PROGRAM MODE_SELECTION_1
VAR
	//MagnetState : (FULL_SHUTDOWN, IDLE, READY_TO_CHARGE, CHARGING, CHARGING_PAUSED, READY_TO_SHOOT, SHOOTING, POST_SHOT, SHUTDOWN, DUMPING); 
	eMagState : E_MagState := 0;
	//bChargingDone: BOOL;
	eCommand : E_Command; // Requested State (FULL_SHUT_DOWN = 0, IDLE = 1, CHARGE = 2, CHARGE_PAUSED, SHOOT = 3, POST_SHOT = 4, SHUTDOWN = 5, DUMPING = 6)
	eStatus : E_Status; // Actual Status (FULL_SHUTDOWN = 0, IDLE = 1, READY_TO_CHARGE = 2, CHARGE = 3, CHARGE_PAUSED = 4, READY_TO_SHOOT = 5, SHOOTING = 6, POST_SHOT = 7, SHUTDOWN = 8, DUMPING = 9, TRIPPED = 10, MANUAL_MODE = 11)
	i: INT;
	
	ChargerOFF_ChrgRlyOPEN_Delay_FShutDown_TON	: TON;
	timerBTW_ChrgRly_ChrgEnable_ChrgPause_TON	: TON;
	timerBTW_ChrgRly_ChrgEnable_ReadyToShoot_TON: TON;
	
	timerBTW_ChrgRly_ChrgEnable_Chrging_TON		: TON;
	timerBTW_ChrgRly_ChrgEnable_PT 	: TIME := T#500MS;
	timerBTW_ChrgRly_ChrgEnable_ET  : TIME;
	
	timerBTW_DUMP_IDLE 				: TON;
	timerBTW_DUMP_IDLE_PT 			: TIME := T#15S;
	timerBTW_DUMP_IDLE_ET 			: TIME;
	
	timerForChargertoTurnOn_TON		: TON;
	timerForChargertoTurnOn_PT		: TIME := T#10S;
	timerForChargertoTurnOn_ET		: TIME;
	ChargersReady					: BOOL;
	
	timerBTW_Shoot_PostShot_TON		: TON;
	timerBTW_Shoot_PostShot_PT      : TIME := T#2S;
	timerBTW_Shoot_PostShot_ET		: TIME;
	
	timerBTW_ChrgEnable_ChrgRly_ShutDown_TON	: TON;
	timerBTW_ChrgEnable_ChrgRly_PT				: TIME := T#1S;
	timerBTW_ChrgEnable_ChrgRly_ET				: TIME;
	
	timerBTW_ChrgEnable_ChrgRly_Dumping_TON		: TON;
	timerBTW_ChrgEnable_ChrgRly_Dumping_ET		: TIME;
	
	timerBTW_ChrgEnable_ChrgRly_Tripped_TON		: TON;
	timerBTW_ChrgEnable_ChrgRly_Tripped_ET		: TIME;
	
	ReadyToChargeRunOutTMR_TON					: TON;
	ReadyToChargeRunOutTMR_PT					: TIME := T#1200S;
	ReadyToChargeRunOutTMR_ET					: TIME;
	
	ChargePausedRunOutTMR_TON					: TON;
	ChargePausedRunOutTMR_PT					: TIME := T#30S;
	ChargePausedRunOutTMR_ET					: TIME;
	
	ReadyToShootRunOutTMR_TON					: TON;
	ReadyToShootRunOutTMR_PT					: TIME := T#60S;
	ReadyToShootRunOutTMR_ET					: TIME;
	
	ShootingRunOutTMR_TON						: TON;
	ShootingRunOutTMR_PT						: TIME := T#3S;
	ShootingRunOutTMR_ET						: TIME;
	
	PostShotRunOutTMR_TON						: TON;
	PostShotRunOutTMR_PT						: TIME := T#2S;
	PostShotRunOutTMR_ET						: TIME;
	
	DumpingRunOutTMR_TON						: TON;
	DumpingRunOutTMR_PT							: TIME := T#300S;
	DumpingRunOutTMR_ET							: TIME;
	
	ChargingRunOutTMR_TON						: TON;
	ChargingRunOutTMR_PT						: TIME := T#600S;
	ChargingRunOutTMR_ET						: TIME;
	
	stControl									: ST_Control;
END_VAR


//LCP Indicator for charged/charging
FOR i := 1 TO 10 BY 1 DO
	IF ( Devices.Coil[i].ChargeRelay_closed = TRUE AND 
		Devices.Coil[i].CoilEnabled = TRUE AND 
		Devices.Coil[i].enableOutputToCharger = TRUE ) OR Devices.Coil[i].ChargeVoltageFeedback >= 10
	THEN
		Devices.Coil[i].SystemCharging := TRUE;
		ELSE
			Devices.Coil[i].SystemCharging := FALSE;
	END_IF;
END_FOR;

//IF any one of the systems is charging or charge, then all system discharge is false, otherwise true
IF Devices.Coil[i].SystemCharging = TRUE THEN
	GVL.AllSystemsDischarged := FALSE;
ELSE
	GVL.AllSystemsDischarged := TRUE;
END_IF;

// IF system is tripped at anytime, it goes to tripped state
IF Trips_DB.SystemTripped = TRUE OR Permissives_DB.SafetyOK = FALSE THEN
	eMagState := E_MagState.TRIPPED;
END_IF;

IF MCP_IO.RemoteModeSelected = FALSE OR HMI_DB.RemoteModeSelected = FALSE THEN  //change auto to remote / manu to local
	eStatus := E_Status.MANUAL_MODE;
END_IF

//At any point, if screen room ask to dump, it goes to dump state
IF (MCP_IO.RemoteModeSelected = TRUE AND eCommand = E_Command.DUMP) OR stControl.Abort = TRUE THEN
	eMagState := E_Magstate.DUMPING;
END_IF;

FOR i := 1 TO 10 BY 1 DO
	Devices.Coil[i].NumOfCap := Tx_Config.CoilSP[i].SysParameters.NumOfCaps;
END_FOR


//Process Starts
CASE eMagState OF 
	//Full Shutdown
	E_MagState.FULL_SHUTDOWN:
						//Disable all Chargers
						FOR i := 1 TO 10 BY 1 DO
							
							//open (de-energize) all interlock relays
							Devices.Coil[i].CloseACInterlockRly := FALSE;
							Devices.Coil[i].enableOutputToCharger := FALSE;
			
							//Close (de-energize) All Dump relays
							Devices.Coil[i].OpenDumpRelays := FALSE;
							
							Devices.Coil[i].CloseHVisolationRelay := FALSE;   //Open all HV isolation relays
						END_FOR;
						
						ChargerOFF_ChrgRlyOPEN_Delay_FShutDown_TON (IN:=TRUE, PT:= timerBTW_ChrgRly_ChrgEnable_PT);
						//delay 500ms before opening charge relay
						IF ChargerOFF_ChrgRlyOPEN_Delay_FShutDown_TON.Q = TRUE THEN
							FOR i := 1 TO 10 BY 1 DO		
							//open (de-energize) all interlock relays
							Devices.Coil[i].closeChargeRelay := FALSE;	
							END_FOR;
							ChargerOFF_ChrgRlyOPEN_Delay_FShutDown_TON (IN:=FALSE, PT:= timerBTW_ChrgRly_ChrgEnable_PT);
						END_IF;
						
						//send shutdown status to screen room
						eStatus := E_Status.FULL_SHUTDOWN;
						//if auto mode selected or hmi automode is selected and screen room asks for idle mode go to idle mode
						IF (MCP_IO.RemoteModeSelected = TRUE OR HMI_DB.RemoteModeSelected = TRUE) AND eCommand = E_Command.IDLE THEN //Auto mode
							GVL.fullshutdown_to_idle := TRUE;
							//if in manu mode and safety is okay and HMI idle MODE PB is pressed, go to idle mode
						ELSIF HMI_DB.RemoteModeSelected = FALSE AND Permissives_DB.SafetyOK = TRUE AND HMI_DB.Idle_mode = TRUE THEN //Manu mode
							GVL.fullshutdown_to_idle := TRUE;
						ELSE
							GVL.fullshutdown_to_idle := FALSE; // otherwise do nothing.
						END_IF;
	
						IF GVL.fullshutdown_to_idle = TRUE THEN
							eMagState := E_MagState.IDLE;
						END_IF;
						//reset all run out tmr
						ReadyToChargeRunOutTMR_TON (IN := FALSE, PT := ReadyToChargeRunOutTMR_PT, ET=>ReadyToChargeRunOutTMR_ET);
						ChargingRunOutTMR_TON (IN := FALSE, PT := ChargingRunOutTMR_PT, ET => ChargingRunOutTMR_ET);
						ChargePausedRunOutTMR_TON (IN := FALSE, PT := ChargePausedRunOutTMR_PT, ET=> ChargePausedRunOutTMR_ET);
						ReadyToShootRunOutTMR_TON (IN := FALSE, PT := ReadyToShootRunOutTMR_PT, ET => ReadyToShootRunOutTMR_ET);
						ShootingRunOutTMR_TON (IN := FALSE, PT := ShootingRunOutTMR_PT, ET => ShootingRunOutTMR_ET);
						PostShotRunOutTMR_TON (IN := FALSE, PT := PostShotRunOutTMR_PT, ET => PostShotRunOutTMR_ET);
						DumpingRunOutTMR_TON (IN := FALSE, PT := DumpingRunOutTMR_PT, ET => DumpingRunOutTMR_ET);
		
	//IDLE STATE
	E_MagState.IDLE:
						eStatus := E_Status.IDLE; //Send status state to screen room
						GVL.dump_to_idle := FALSE;
						//reset all run out tmr
						ReadyToChargeRunOutTMR_TON (IN := FALSE, PT := ReadyToChargeRunOutTMR_PT, ET=>ReadyToChargeRunOutTMR_ET);
						ChargingRunOutTMR_TON (IN := FALSE, PT := ChargingRunOutTMR_PT, ET => ChargingRunOutTMR_ET);
						ChargePausedRunOutTMR_TON (IN := FALSE, PT := ChargePausedRunOutTMR_PT, ET=> ChargePausedRunOutTMR_ET);
						ReadyToShootRunOutTMR_TON (IN := FALSE, PT := ReadyToShootRunOutTMR_PT, ET => ReadyToShootRunOutTMR_ET);
						ShootingRunOutTMR_TON (IN := FALSE, PT := ShootingRunOutTMR_PT, ET => ShootingRunOutTMR_ET);
						PostShotRunOutTMR_TON (IN := FALSE, PT := PostShotRunOutTMR_PT, ET => PostShotRunOutTMR_ET);
						DumpingRunOutTMR_TON (IN := FALSE, PT := DumpingRunOutTMR_PT, ET => DumpingRunOutTMR_ET);
						
						// Local MODE
						IF (MCP_IO.RemoteModeSelected = FALSE OR HMI_DB.RemoteModeSelected = FALSE)AND 
							HMI_DB.chargePB = TRUE AND 
							Permissives_DB.SafetyOK = TRUE AND 
							GVL.AllSystemsDischarged = TRUE 
							THEN   
								//open dump relays
								FOR i := 1 TO 10 BY 1 DO
									Devices.Coil[i].OpenDumpRelays := TRUE; //NC contact
								END_FOR;
			
								GVL.idle_to_readyToCharge := TRUE;
							ELSE
								GVL.idle_to_readyToCharge := FALSE;
						END_IF;
						//Remote MODE
						// ready to go to charge state when dump relays are all open and charge permissive is satisfied 
						IF (MCP_IO.RemoteModeSelected = TRUE OR HMI_DB.RemoteModeSelected = TRUE) AND 
							Permissives_DB.SafetyOK = TRUE AND GVL.AllSystemsDischarged = TRUE
							THEN 
								//open dump relays
								FOR i := 1 TO 10 BY 1 DO
									Devices.Coil[i].OpenDumpRelays := TRUE; //NC contact
								END_FOR;	
								GVL.idle_to_readyToCharge := TRUE;
						ELSE
							GVL.idle_to_readyToCharge := FALSE;
							//Keep dump relays close if no command to go to charging state
							FOR i := 1 TO 10 BY 1 DO
								Devices.Coil[i].OpenDumpRelays := FALSE; //NC contact
							END_FOR;
						END_IF;
		
						IF GVL.idle_to_readyToCharge = TRUE AND Permissives_DB.ChargePermOK = TRUE AND GVL.AllSystemsDischarged = TRUE THEN
							eMagState := E_MagState.READY_TO_CHARGE;
						ELSIF (MCP_IO.RemoteModeSelected = TRUE AND eCommand = E_Command.FULL_SHUTDOWN) 
							THEN 
								eMagState := E_MagState.FULL_SHUTDOWN;
						END_IF;
						
	//Charging State	
	E_MagState.READY_TO_CHARGE:
						//reset bit
						GVL.idle_to_readyToCharge := FALSE;
						//send status to screenroom
						eStatus := E_Status.READY_TO_CHARGE;
						
						ReadyToChargeRunOutTMR_TON (IN := TRUE, PT := ReadyToChargeRunOutTMR_PT, ET=>ReadyToChargeRunOutTMR_ET);
						IF ReadyToChargeRunOutTMR_TON.Q = TRUE THEN
							Trips_DB.MachineTimedOut := TRUE;
							eMagState := E_MagState.TRIPPED;
							ReadyToChargeRunOutTMR_TON (IN := FALSE, PT := ReadyToChargeRunOutTMR_PT, ET=>ReadyToChargeRunOutTMR_ET);
						END_IF
						
						IF Permissives_DB.ChargePermOK = TRUE AND 
							MCP_IO.RemoteModeSelected = TRUE AND 
							eCommand = E_Command.CHARGE 
							THEN
								eMagState := E_MagState.CHARGING;
						ELSIF (MCP_IO.RemoteModeSelected = TRUE AND eCommand = E_Command.FULL_SHUTDOWN) 
							THEN 
								eMagState := E_MagState.FULL_SHUTDOWN;
						END_IF;
					
	//Charging State	
	E_MagState.CHARGING:	
						//send charging status to screen room
						eStatus := E_Status.CHARGING;
						
						ChargingRunOutTMR_TON (IN := TRUE, PT := ChargingRunOutTMR_PT, ET => ChargingRunOutTMR_ET);
						IF ChargingRunOutTMR_TON.Q = TRUE THEN
							Trips_DB.MachineTimedOut := TRUE;
							eMagState := E_MagState.TRIPPED;
							ChargingRunOutTMR_TON (IN := FALSE, PT := ChargingRunOutTMR_PT, ET => ChargingRunOutTMR_ET);
						END_IF
						
						IF Permissives_DB.SafetyOK THEN
						//Close all AC interlock contactor
							FOR i := 1 TO 10 BY 1 DO	
								Devices.Coil[i].CloseACInterlockRly := TRUE;
							END_FOR;
						END_IF;
	
						IF Permissives_DB.SafetyOK = TRUE AND MCP_IO.RemoteModeSelected = TRUE AND HMI_DB.StopPB = FALSE THEN
						//Close all Charge Relays
							FOR i := 1 TO 10 BY 1 DO	
								Devices.Coil[i].closeChargeRelay := TRUE;	
							END_FOR;	
						END_IF;
						
						IF Permissives_DB.AllChargerRelay_Closed = TRUE THEN
							//wait 500ms before turning on chargers
							timerBTW_ChrgRly_ChrgEnable_Chrging_TON (IN := TRUE, PT := timerBTW_ChrgRly_ChrgEnable_PT, ET => timerBTW_ChrgRly_ChrgEnable_ET);
							IF timerBTW_ChrgRly_ChrgEnable_Chrging_TON.Q = TRUE THEN 
								FOR i := 1 TO 10 BY 1 DO	
									Devices.Coil[i].enableOutputToCharger := TRUE;  //turn on all chargers	
								END_FOR;
							END_IF;	
							timerBTW_ChrgRly_ChrgEnable_Chrging_TON (IN := FALSE, PT := timerBTW_ChrgRly_ChrgEnable_PT, ET => timerBTW_ChrgRly_ChrgEnable_ET);
						ELSE 
							eMagState := E_MagState.DUMPING;
						END_IF;
	
						IF Permissives_DB.AllChargerEnabled = TRUE AND Permissives_DB.AlldcPSUok = TRUE THEN 
							//wait 10sec before setting the setpoint (Darren's sequence)
							timerForChargertoTurnOn_TON (IN := TRUE, PT := timerForChargertoTurnOn_PT, ET => timerForChargertoTurnOn_ET);
			
							IF timerForChargertoTurnOn_TON.Q = TRUE THEN
								//ChargersReady := TRUE;
								FOR i := 1 TO 10 BY 1 DO	
									Devices.Coil[i].currentSetpoint := Setpoints.Coil[i].RecipeLocal.currentSetpoint;	//setpoints from recipe	
									Devices.Coil[i].chargerSetpoint := Setpoints.Coil[i].RecipeLocal.chargerSetpoint;	//setpoints from recipe		
								END_FOR;
								timerForChargertoTurnOn_TON (IN := FALSE);
							END_IF;	
						ELSE 
							timerForChargertoTurnOn_TON (IN := FALSE);
						END_IF;
						
						// IF in manual mode and HMI pause pb is pressed | in auto mode and command from screenroom goes to pause charge, go to pause charge mode.
						IF (HMI_DB.PausePB AND MCP_IO.RemoteModeSelected = FALSE) THEN
							eMagState := E_MagState.CHARGE_PAUSED;
						END_IF;
						
						// IF in manual mode, Dump PB is pressed, go to dump mode, IF auto mode is selected, and command from screen room asks to dump go to dump mode.
						IF (HMI_DB.dumpPB = TRUE AND MCP_IO.RemoteModeSelected = FALSE) OR (MCP_IO.RemoteModeSelected = TRUE AND eCommand = E_Command.DUMP) THEN 
							eMagState := E_magState.DUMPING;
						END_IF;
						
						// if ultracap over voltage go to charge paused 
						IF Devices.Coil[i].CapWarning = TRUE THEN
							eMagState := E_MagState.CHARGE_PAUSED;
						END_IF;
						
						//IF Cap voltage = charger voltages is reached, Ready_TO_SHOOT  _ need to be recipe user input voltage
						
						IF Permissives_DB.AllCoilCapsCharged = TRUE AND GVL.AllChargerReadywithSP = TRUE
							THEN
								GVL.charge_to_readyToShoot := TRUE;
							ELSE
								GVL.charge_to_readyToShoot := FALSE;
						END_IF;
						
						IF GVL.charge_to_readyToShoot = TRUE THEN
							eMagState := E_MagState.READY_TO_SHOOT;	
							timerForChargertoTurnOn_TON (IN := FALSE, PT := timerForChargertoTurnOn_PT);
						END_IF;
		
	//Charge Paused State	
	E_MagState.CHARGE_PAUSED:
						// send status to screen room
						eStatus := E_Status.CHARGING_PAUSED;
						//Start RUNout timer
						ChargePausedRunOutTMR_TON (IN := TRUE, PT := ChargePausedRunOutTMR_PT, ET=> ChargePausedRunOutTMR_ET);// Recipe.General.ChargeRunOutTime);
						
						//Turn on disable charger
						FOR i := 1 TO 10 BY 1 DO
							Devices.Coil[i].enableOutputToCharger := FALSE;
						END_FOR;
						//wait 500ms
						timerBTW_ChrgRly_ChrgEnable_ChrgPause_TON (IN := TRUE, PT := timerBTW_ChrgEnable_ChrgRly_PT, ET => timerBTW_ChrgEnable_ChrgRly_ET);
						
						//open charger relay
						IF timerBTW_ChrgRly_ChrgEnable_ChrgPause_TON.Q = TRUE THEN
							FOR i := 1 TO 10 BY 1 DO
								Devices.Coil[i].closeChargeRelay := FALSE;
							END_FOR;
							timerBTW_ChrgRly_ChrgEnable_ChrgPause_TON (IN := FALSE, PT := timerBTW_ChrgRly_ChrgEnable_PT);
						END_IF
						IF HMI_DB.StopPB = TRUE OR (MCP_IO.RemoteModeSelected AND Permissives_DB.SafetyOK = FALSE) THEN 
							eMagState := E_MagState.DUMPING;	
						END_IF;
			
						//IF CANBus Warning/fault goes away, go back to charging
					
						IF (Devices.Coil[1].CapWarning = FALSE OR Devices.Coil[1].CoilEnabled = FALSE) AND
							(Devices.Coil[2].CapWarning = FALSE OR Devices.Coil[2].CoilEnabled = FALSE) AND
							(Devices.Coil[3].CapWarning = FALSE OR Devices.Coil[3].CoilEnabled = FALSE) AND
							(Devices.Coil[4].CapWarning = FALSE OR Devices.Coil[4].CoilEnabled = FALSE) AND
							(Devices.Coil[5].CapWarning = FALSE OR Devices.Coil[5].CoilEnabled = FALSE) AND
							(Devices.Coil[6].CapWarning = FALSE OR Devices.Coil[6].CoilEnabled = FALSE) AND
							(Devices.Coil[7].CapWarning = FALSE OR Devices.Coil[7].CoilEnabled = FALSE) AND
							(Devices.Coil[8].CapWarning = FALSE OR Devices.Coil[8].CoilEnabled = FALSE) AND
							(Devices.Coil[9].CapWarning = FALSE OR Devices.Coil[9].CoilEnabled = FALSE) AND
							(Devices.Coil[10].CapWarning = FALSE OR Devices.Coil[10].CoilEnabled = FALSE) 
						THEN
							eMagState := E_MagState.CHARGING;
						END_IF;
						
						//When RUNout timer runs out, and still in shooting state, trip the system
						IF ChargePausedRunOutTMR_TON.Q THEN
							Trips_DB.MachineTimedOut := TRUE;
							eMagState := E_MagState.TRIPPED;
							//reset timer
							ChargePausedRunOutTMR_TON (IN := FALSE, PT := ChargePausedRunOutTMR_PT, ET=> ChargePausedRunOutTMR_ET);
						END_IF;
 
						
	 E_MagState.READY_TO_SHOOT:
	 
						GVL.charge_to_readyToShoot := FALSE;
						
						//Start RUNout timer
						ReadyToShootRunOutTMR_TON (IN := TRUE, PT := ReadyToShootRunOutTMR_PT, ET => ReadyToShootRunOutTMR_ET);
						
						IF GVL.AllChargerReadywithSP = FALSE THEN
							eMagState := E_MagState.CHARGING;
						END_IF
						
						//when it is ready to shoot, disable chargers
						FOR i := 1 TO 10 BY 1 DO
							Devices.Coil[i].enableOutputToCharger := FALSE;
						END_FOR;
						//wait 500ms
						timerBTW_ChrgRly_ChrgEnable_ReadyToShoot_TON (IN := TRUE, PT := timerBTW_ChrgRly_ChrgEnable_PT, ET => timerBTW_ChrgRly_ChrgEnable_ET);
						
						//open all charger relays and AC interlock relays
						IF timerBTW_ChrgRly_ChrgEnable_ReadyToShoot_TON.Q = TRUE THEN
							FOR i := 1 TO 10 BY 1 DO
								Devices.Coil[i].closeChargeRelay := FALSE;
								Devices.Coil[i].CloseACInterlockRly := FALSE;
								//set current setpoint 
								Devices.Coil[i].currentSetpoint := Setpoints.Coil[i].RecipeLocal.currentSetpoint;
							END_FOR;
							timerBTW_ChrgRly_ChrgEnable_ReadyToShoot_TON (IN := FALSE);
						END_IF;
						
						IF Trips_DB.SystemTripped = FALSE AND Permissives_DB.ShootPermOK = TRUE THEN
							eStatus := E_Status.READY_TO_SHOOT;  //send status to screen room
							GVL.readyToShoot_to_Shoot := TRUE;
						ELSIF (Trips_DB.SystemTripped = TRUE OR Permissives_DB.ShootPermOK = FALSE OR eCommand = E_Command.DUMP) THEN
							GVL.readyToShoot_to_Shoot := FALSE;
							eMagState := E_MagState.DUMPING;
						END_IF;

						IF GVL.readyToShoot_to_Shoot = TRUE AND eCommand = E_Command.SHOOT THEN
			
							eMagState := E_MagState.SHOOTING;
						END_IF;
						
						IF MCP_IO.RemoteModeSelected = TRUE AND eCommand = E_Command.FULL_SHUTDOWN THEN
							GVL.readyToShoot_to_Shoot := FALSE;
							eMagState := E_MagState.FULL_SHUTDOWN;
						END_IF;
						
						//When RUNout timer runs out, and still in shooting state, trip the system
						IF ReadyToShootRunOutTMR_TON.Q THEN
							Trips_DB.MachineTimedOut := TRUE;
							eMagState := E_MagState.TRIPPED;
							//reset timer
							ReadyToShootRunOutTMR_TON (IN := FALSE, PT := ReadyToShootRunOutTMR_PT, ET => ReadyToShootRunOutTMR_ET);
						END_IF;
		
	E_MagState.SHOOTING:
	 					// turn off the readyToShoot_TO_Shoot bit 
						GVL.readyToShoot_to_Shoot := FALSE;
						
						//report shooting state to screen room
						eStatus := E_Status.SHOOTING;
						
						ShootingRunOutTMR_TON (IN := TRUE, PT := ShootingRunOutTMR_PT, ET => ShootingRunOutTMR_ET);
						
						FOR i := 1 TO 10 BY 1 DO
							Devices.Coil[i].CloseHVisolationRelay := TRUE;
						END_FOR;
						
						//send current feedback to screenroom, something :=  Devices.Coil[i].CurrentFeedback; ????
						
						//if screen room ask to dump, or in manual mode and stopPB or dumpPB is pressed go to dump mode
						IF eCommand = E_Command.DUMP OR (MCP_IO.RemoteModeSelected = FALSE AND (HMI_DB.dumpPB= TRUE OR HMI_DB.StopPB = TRUE)) THEN
							eMagState := E_MagState.DUMPING;
						END_IF;
						
						timerBTW_Shoot_PostShot_TON (IN := TRUE, PT := timerBTW_Shoot_PostShot_PT, ET=> timerBTW_Shoot_PostShot_ET);
				
						IF timerBTW_Shoot_PostShot_TON.Q = TRUE THEN
							GVL.shoot_to_postShot := TRUE;
							timerBTW_Shoot_PostShot_TON (IN := FALSE, PT := timerBTW_Shoot_PostShot_PT, ET=> timerBTW_Shoot_PostShot_ET);
							ELSE
								GVL.shoot_to_postShot := FALSE;
						END_IF;
						
						IF Trips_DB.SystemTripped = FALSE THEN	
							GVL.shot_going_OK := TRUE;
							ELSE
								GVL.shot_going_OK := FALSE;
						END_IF;
						
						IF GVL.shoot_to_postShot = TRUE AND GVL.shot_going_OK = TRUE THEN
							eMagState := E_MagState.POST_SHOT;
							ELSE IF ShootingRunOutTMR_TON.Q = TRUE THEN 
								Trips_DB.MachineTimedOut := TRUE;
								eMagState := E_MagState.TRIPPED;
								ShootingRunOutTMR_TON (IN := FALSE, PT := ShootingRunOutTMR_PT, ET => ShootingRunOutTMR_ET);
							END_IF
						END_IF;		
		
	E_MagState.POST_SHOT:
						GVL.shoot_to_postShot := FALSE;
						
						PostShotRunOutTMR_TON (IN := TRUE, PT := PostShotRunOutTMR_PT, ET => PostShotRunOutTMR_ET);
						
						//Send status to screenroom
						eStatus := E_Status.POST_SHOT;
						//open HV isolation Relays
						FOR i := 1 TO 10 BY 1 DO
							Devices.Coil[i].CloseHVisolationRelay := FALSE;
						END_FOR;
						
						//if temperature are all good and safety is okay, shot is done
						IF Permissives_DB.SafetyOK = TRUE AND Devices.Coil[i].ChargeVoltageFeedback <= 10 THEN
							GVL.shot_is_done := TRUE;
							ELSE
								GVL.shot_is_done := FALSE;
						END_IF;
						
						//if shot is done, go back to idle state  // it was shot is done or command.idle
						IF GVL.shot_is_done = TRUE AND (MCP_IO.RemoteModeSelected = TRUE AND eCommand = E_Command.IDLE) THEN
							eMagState := E_MagState.IDLE;
						//if screen room ask to dump, or in manual mode and stopPB or dumpPB is pressed go to dump mode
						ELSIF eCommand = E_Command.DUMP OR (MCP_IO.RemoteModeSelected = FALSE AND (HMI_DB.dumpPB= TRUE OR HMI_DB.StopPB = TRUE)) THEN
							eMagState := E_MagState.DUMPING;
						ELSIF (MCP_IO.RemoteModeSelected = TRUE AND eCommand = E_Command.FULL_SHUTDOWN) THEN 
							eMagState := E_MagState.FULL_SHUTDOWN;
						END_IF;
						
						IF PostShotRunOutTMR_TON.Q = TRUE THEN
							Trips_DB.MachineTimedOut := TRUE;
							eMagState := E_MagState.TRIPPED;
							PostShotRunOutTMR_TON (IN := FALSE, PT := PostShotRunOutTMR_PT, ET => PostShotRunOutTMR_ET);
						END_IF
								
	E_MagState.DUMPING:	
						//disable all chargers
						FOR i := 1 TO 10 BY 1 DO
							Devices.Coil[i].enableOutputToCharger := FALSE;
							Devices.Coil[i].CloseHVisolationRelay := FALSE;   //Open all HV isolation relays
						END_FOR
						
						IF Permissives_DB.AllChargerEnabled = FALSE THEN 
							timerBTW_ChrgEnable_ChrgRly_Dumping_TON (IN := TRUE, PT := timerBTW_ChrgRly_ChrgEnable_PT, ET=>timerBTW_ChrgEnable_ChrgRly_Dumping_ET); 					 
						ELSE
							timerBTW_ChrgEnable_ChrgRly_Dumping_TON (IN := FALSE);
						END_IF;
						
						IF timerBTW_ChrgEnable_ChrgRly_Dumping_TON.Q = TRUE THEN
							FOR i := 1 TO 10 BY 1 DO
								Devices.Coil[i].closeChargeRelay := FALSE; //open charge relay
							END_FOR;
							timerBTW_ChrgEnable_ChrgRly_Dumping_TON (IN := FALSE);
						END_IF;
						
						//Close all dump relays
						Devices.Coil[1].OpenDumpRelays := FALSE; //NC so close dump relays
						Devices.Coil[2].OpenDumpRelays := FALSE;
						Devices.Coil[3].OpenDumpRelays := FALSE;
						Devices.Coil[4].OpenDumpRelays := FALSE;
						Devices.Coil[5].OpenDumpRelays := FALSE;
						Devices.Coil[6].OpenDumpRelays := FALSE;
						Devices.Coil[7].OpenDumpRelays := FALSE;
						Devices.Coil[8].OpenDumpRelays := FALSE;
						Devices.Coil[9].OpenDumpRelays := FALSE;
						Devices.Coil[10].OpenDumpRelays := FALSE;
						
						//send state to screen room
						eStatus := E_Status.DUMPING;
						
						DumpingRunOutTMR_TON (IN := TRUE, PT := DumpingRunOutTMR_PT, ET => DumpingRunOutTMR_ET);
						IF DumpingRunOutTMR_TON.Q = TRUE THEN
							Trips_DB.MachineTimedOut := TRUE;
							eMagState := E_MagState.TRIPPED;
							DumpingRunOutTMR_TON (IN := FALSE, PT := DumpingRunOutTMR_PT, ET => DumpingRunOutTMR_ET);
						END_IF
						
						//NC, if all dump relays are closed, and all cap voltage discharged, start timer and go back to IDLE automaticlally
						IF Permissives_DB.AllDumpRelayOpen = FALSE AND Permissives_DB.AllCoilCapsCharged = FALSE THEN 
							timerBTW_DUMP_IDLE (IN := TRUE, PT := timerBTW_DUMP_IDLE_PT, ET => timerBTW_DUMP_IDLE_ET);
							IF timerBTW_DUMP_IDLE.Q = TRUE THEN 
								GVL.dump_to_idle := TRUE;
							END_IF;	
						ELSE
							timerBTW_DUMP_IDLE (IN := FALSE);
							GVL.dump_to_idle := FALSE;	
						END_IF;
						
						IF GVL.dump_to_idle = TRUE THEN
							eMagState := E_MagState.IDLE;
							timerBTW_DUMP_IDLE (IN := FALSE, PT := timerBTW_DUMP_IDLE_PT);
						ELSIF GVL.dump_to_idle = TRUE AND MCP_IO.RemoteModeSelected = TRUE AND eCommand = E_Command.FULL_SHUTDOWN THEN
								eMagState := E_MagState.FULL_SHUTDOWN;
						END_IF;
						//GVL.dump_to_idle := FALSE;
						
	E_MagState.TRIPPED: 
						eStatus := E_Status.TRIPPED;	
						
						FOR i := 1 TO 10 BY 1 DO
							//Disable all Chargers
							Devices.Coil[i].enableOutputToCharger := FALSE;
		
							//open (de-energize) all interlock relays
							Devices.Coil[i].CloseACInterlockRly := FALSE;
	
							//Close (de-energize) All Dump relays
							Devices.Coil[i].OpenDumpRelays := FALSE;
							
							Devices.Coil[i].CloseHVisolationRelay := FALSE;   //Open all HV isolation relays
						END_FOR;
						//wait 500ms before opening the charge relay
						timerBTW_ChrgEnable_ChrgRly_Tripped_TON (IN := TRUE, PT := timerBTW_ChrgEnable_ChrgRly_PT, ET => timerBTW_ChrgEnable_ChrgRly_Tripped_ET);
						
						IF timerBTW_ChrgEnable_ChrgRly_Tripped_TON.Q = TRUE THEN
							FOR i := 1 TO 10 BY 1 DO
							//open all charge relays
							Devices.Coil[i].closeChargeRelay := FALSE;
							END_FOR;
							timerBTW_ChrgEnable_ChrgRly_Tripped_TON (IN := FALSE, PT := timerBTW_ChrgEnable_ChrgRly_PT, ET => timerBTW_ChrgEnable_ChrgRly_Tripped_ET);
						END_IF;
						
						// when Trip is clear by the opeartor, it goes back to idle state.
						IF Trips_DB.SystemTripped = FALSE AND Permissives_DB.SafetyOK = TRUE THEN 
							eMagState := E_MagState.IDLE;
						END_IF;
						
						//reset all run out tmr
						ReadyToChargeRunOutTMR_TON (IN := FALSE, PT := ReadyToChargeRunOutTMR_PT, ET=>ReadyToChargeRunOutTMR_ET);
						ChargingRunOutTMR_TON (IN := FALSE, PT := ChargingRunOutTMR_PT, ET => ChargingRunOutTMR_ET);
						ChargePausedRunOutTMR_TON (IN := FALSE, PT := ChargePausedRunOutTMR_PT, ET=> ChargePausedRunOutTMR_ET);
						ReadyToShootRunOutTMR_TON (IN := FALSE, PT := ReadyToShootRunOutTMR_PT, ET => ReadyToShootRunOutTMR_ET);
						ShootingRunOutTMR_TON (IN := FALSE, PT := ShootingRunOutTMR_PT, ET => ShootingRunOutTMR_ET);
						PostShotRunOutTMR_TON (IN := FALSE, PT := PostShotRunOutTMR_PT, ET => PostShotRunOutTMR_ET);
						DumpingRunOutTMR_TON (IN := FALSE, PT := DumpingRunOutTMR_PT, ET => DumpingRunOutTMR_ET);
						
END_CASE

//run hmi 
HMI();

//reset counter
IF i > 10 THEN 
	i := 1;
END_IF;

END_PROGRAM

(* stored: Version 1.1.0.1, ProductVersion 3.1.4024.11
   POU MODE_SELECTION_1: Id {555b4fc9-29ab-4725-aacb-810ee58c0cd6}, SpecialFunc None *)
